FUNCTION_BLOCK FB_Interval
VAR_INPUT
	bInterval:BOOL;
	ET_Current:Time;
	Pressed:BOOL:=FALSE;
	cInterval:INT:=0;
END_VAR
VAR_OUTPUT
	Intervals: ARRAY[1..20] OF TIME;
	
END_VAR
VAR
	i:INT;
	

END_VAR

IF bInterval AND  Pressed THEN
	cInterval:=cInterval + 1;
	bInterval:=FALSE;
	Pressed:=false;
	
	
	IF cInterval > 20 THEN
		cInterval:=20;
		FOR i:=1 TO 19 DO 
			Intervals[i]:=Intervals[i+1];
			
		END_FOR
	END_IF
	Intervals[cInterval]:=ET_Current;
END_IF

END_FUNCTION_BLOCK

(* stored: Version 1.1.0.1, ProductVersion 3.1.4026.8
   POU FB_Interval: Id {b5f63a85-0ecb-4507-902a-f3cb0580e823}, SpecialFunc None *)
